// TIA Portal V20 program export: 1 tag tables, 0 data types, 0 data blocks, 1 code blocks (in call order from the OBs), 0 instance data blocks

VAR_GLOBAL   // PLC tag table "Default tag table"
   ent_uno AT %I0.0 : Bool;
   sal_uno AT %Q0.0 : Bool;
   Tag_1 AT %M50.0 : Bool;
   Tag_2 AT %M50.2 : Bool;
   Tag_3 AT %M50.6 : Bool;
END_VAR

ORGANIZATION_BLOCK "Main"   // OB1, LAD, ProgramCycle
TITLE = "Main Program Sweep (Cycle)"
{ S7_Optimized_Access := 'TRUE' }
// stored: SetENOAutomatically false
   VAR_INPUT
      Initial_Call : Bool;   // Initial call of this OB
      Remanence : Bool;   // =True, if remanent data are available
   END_VAR
BEGIN

REGION Network 1
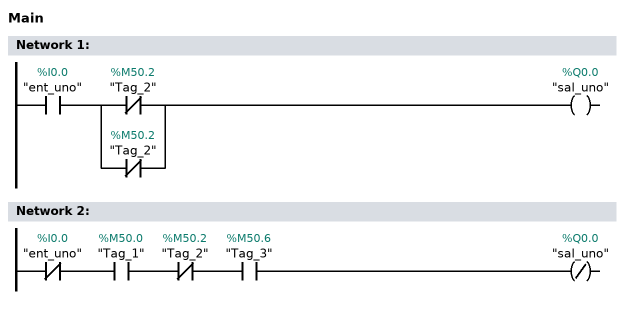
   RUNG wire#powerrail
      Contact( "ent_uno" )
      wire#w1
      I_Contact( "Tag_2" )
      wire#w2
      Coil( "sal_uno" )
   END_RUNG
   RUNG wire#w1
      I_Contact( "Tag_2" )
   END_RUNG wire#w2
   // the same network as SCL:
   "sal_uno" := "ent_uno" AND (NOT "Tag_2" OR NOT "Tag_2");
END_REGION

REGION Network 2
   RUNG wire#powerrail
      I_Contact( "ent_uno" )
      Contact( "Tag_1" )
      I_Contact( "Tag_2" )
      Contact( "Tag_3" )
      I_Coil( "sal_uno" )
   END_RUNG
   // the same network as SCL:
   "sal_uno" := NOT (NOT "ent_uno" AND "Tag_1" AND NOT "Tag_2" AND "Tag_3");
END_REGION
END_ORGANIZATION_BLOCK
